FUNCTION_BLOCK FB_HeartBeat_Subsystem
VAR_INPUT
	
END_VAR
VAR_OUTPUT
	heart_timeout_Alarm:BOOL;
END_VAR
VAR
	bReset_ads_heart_beat	: HeartbeatParams;
	bReset_ads_heart_beatTemp	: HeartbeatParams;
	heart_timeout:TON;
	AA: INT;
END_VAR

heart_timeout(PT:=T#3S);

IF bReset_ads_heart_beat.current_time_ms=bReset_ads_heart_beatTemp.current_time_ms THEN
	heart_timeout.IN	:=TRUE;
ELSE
	heart_timeout.IN	:=FALSE;
	heart_timeout_Alarm:=FALSE;
	bReset_ads_heart_beatTemp.current_time_ms	:= bReset_ads_heart_beat.current_time_ms;	
END_IF

IF heart_timeout.Q  THEN
	heart_timeout.IN:=FALSE;
	heart_timeout_Alarm:=TRUE;
END_IF
//heartbeat(bReset_ads_heart_beat);

{attribute 'TcRpcEnable'}
METHOD heartbeat : UDINT
VAR_INPUT
	heartbeat_params : HeartbeatParams;	
END_VAR
heartbeat	:= 1; 
bReset_ads_heart_beat	:= heartbeat_params;
heartbeat	:= MethodCallReturnValue.ACCEPTED;

AA:=AA+1;
END_METHOD

END_FUNCTION_BLOCK

(* stored: Version 1.1.0.1, ProductVersion 3.1.4024.12
   POU FB_HeartBeat_Subsystem: Id {f4705ac8-c2e7-4066-9e2a-39c2c41daf98}, SpecialFunc None
   Method heartbeat: Id {f3dcafaa-9e61-4170-9f3f-99aa20b20ebc} *)
